FUNCTION_BLOCK FB_IOs
VAR_INPUT
END_VAR
VAR_OUTPUT
END_VAR
VAR
END_VAR

{attribute 'TcRpcEnable'}
METHOD Check : BOOL
VAR_INPUT
END_VAR
END_METHOD

END_FUNCTION_BLOCK

(* stored: Version 1.1.0.1, ProductVersion 3.1.4024.11
   POU FB_IOs: Id {4db9a8db-2dbb-495a-ba78-a803ff7bd4d7}, SpecialFunc None
   Method Check: Id {e65b581f-0727-480e-9083-0f7e20a36f9e} *)
